(* IEC 61131-3 sources: Industry-PLC-LLM/data/PLCBEAD_repo/PLCBEAD_PLCEmbed-main/PLC-BEAD/Source/GEB/GEN_BIT, 1 file *)

(* ---- GEN_BIT.ST ---- *)
FUNCTION BIT_OF_DWORD : BOOL
  VAR_INPUT
    IN : DWORD;
    N : INT;
  END_VAR

  BIT_OF_DWORD := (SHR(IN,N) AND 16#00000001) > 0;
END_FUNCTION

FUNCTION_BLOCK GEN_BIT_Block

	VAR_INPUT
		IN0 :	DWORD;
		IN1 :	DWORD;
		IN2 :	DWORD;
		IN3 :	DWORD;
		CLK :	BOOL;
		STEPS :	INT;
		REP :	INT;
		RST :	BOOL;
	END_VAR

	VAR_OUTPUT
		Q0 :	BOOL;
		Q1 :	BOOL;
		Q2 :	BOOL;
		Q3 :	BOOL;
		CNT :	INT;
		RUN :	BOOL;
	END_VAR

	VAR
		r0 :	DWORD;
		R1  :	DWORD;
		R2 :	DWORD;
		r3 :	DWORD;
		rx :	INT := 1;
	END_VAR

	IF CLK AND NOT RST THEN
		RUN := (REP = 0) OR (rx <= REP);
		IF RUN THEN
			IF CNT = STEPS THEN
				CNT := 0;
			END_IF;

			IF CNT = 0 THEN
				r0 := IN0;
				R1  := IN1;
				R2 := IN2;
				r3 := IN3;
			END_IF;

			IF (CNT < STEPS) THEN
				Q0 := BIT_OF_DWORD(r0,0);
				Q1 := BIT_OF_DWORD(R1 ,0);
				Q2 := BIT_OF_DWORD(R2,0);
				Q3 := BIT_OF_DWORD(r3,0);
				r0 := SHR(r0,1);
				R1  := SHR(R1 ,1);
				R2 := SHR(R2,1);
				r3 := SHR(r3,1);
			END_IF;

			CNT := CNT +1;
			IF (CNT = STEPS) AND (REP <> 0) THEN rx := rx +1; END_IF;
			IF (rx > REP) AND (REP <> 0) THEN RUN := FALSE; END_IF;
		END_IF;
	ELSE
		IF RST THEN
			RUN := FALSE;
			Q0 := FALSE;
			Q1 := FALSE;
			Q2 := FALSE;
			Q3 := FALSE;
			r0 := DWORD#0;
			R1  := DWORD#0;
			R2 := DWORD#0;
			r3 := DWORD#0;
			CNT := 0;
			rx := 1;
		END_IF;
	END_IF;

END_FUNCTION_BLOCK

PROGRAM program0
  VAR
	IN0 :	DWORD;
	IN1 :	DWORD;
	IN2 :	DWORD;
	IN3 :	DWORD;
	CLK :	BOOL;
	STEPS :	INT;
	REP :	INT;
	RST :	BOOL;
	Q0 :	BOOL;
	Q1 :	BOOL;
	Q2 :	BOOL;
	Q3 :	BOOL;
	CNT :	INT;
	RUN :	BOOL;
	func_block : GEN_BIT_Block;
  END_VAR
	func_block.IN0  :=IN0;
	func_block.IN1  :=IN1;
	func_block.IN2  :=IN2;
	func_block.IN3  :=IN3;
	func_block.CLK  :=CLK;
	func_block.STEPS  :=STEPS;
	func_block.REP  :=REP;
	func_block.RST  :=RST;
	func_block();
	Q0 := func_block.Q0;
	Q1 := func_block.Q1;
	Q2 := func_block.Q2;
	Q3 := func_block.Q3;
	CNT := func_block.CNT;
	RUN := func_block.RUN;

END_PROGRAM
